(* CODESYS project Trabalho_2.project

Project tree, tasks and I/O mapping:
  Device : CODESYS Control Win V3, 3S - Smart Software Solutions GmbH, order no. 305021, version 3.5.11.30
    application Application
      libraries: Standard, * (System)
      task MainTask (cyclic, interval t#20ms, priority 1) calls PLC_PRG
      program PLC_PRG [LD]
      Symbols
*)

// Device/Application/PLC_PRG
PROGRAM PLC_PRG
VAR
	M0_1: BOOL;
	M0_0: BOOL;
	M0_2: BOOL;
	OCIOSO: BOOL;
	B_ON: BOOL;
	T01: BOOL;
	ET02: BOOL;
	A: BOOL;
	B: BOOL;
	T02: BOOL;
	ET03: BOOL;
	T03: BOOL;
	ET04: BOOL;
	T04: BOOL;
	ET05: BOOL;
	C: BOOL;
	Cont_Blocos: CTU;
	Zera_Cont: BOOL;
	Timer_Roletada: TON;
	TR: TIME;
	VOID: BOOL;
	T05: BOOL;
	T06: BOOL;
	ET06: BOOL;
	E01: BOOL;
	E02: BOOL;
	E03: BOOL;
	EB: BOOL;
	Pist_Retraido: BOOL;
	Presenca_Balanca: BOOL;
	ET07: BOOL;
	PESO: REAL;
	AUXILIAR: BOOL;
	T07: BOOL;
	TIMER_VOID: BOOL;
	T08: BOOL;
	ET08: BOOL;
	TON_0: TON;
	TIMER_TO_SEPARATION: TIME;
	EP: BOOL;
	ET09: BOOL;
	ET10: BOOL;
	ET11: BOOL;
	EM: BOOL;
	PISTAO: BOOL;
	SENSOR_PLASTICO: BOOL;
	T09: BOOL;
	TON_1: TON;
	RESET_PLASTICO: TIME;
	EP_OFF: BOOL;
	T10: BOOL;
	T11: BOOL;
	TON_2: TON;
	RESET_METAL: TIME;
	EM_OFF: BOOL;
	SENSOR_METAL: BOOL;
	VALOR: INT;
	_PESP: REAL;
	TEMPO_09: TON;
	TEMP1: TIME;
	TEMPO_11: TON;
	TEMP2: TIME;
	TIMER_BALANCA: TOF;
	TB: TIME;
	SALARIBA: BOOL;
	TIMER_BALANCA_OFF: TON;
	TIMER_BALAN: TON;
	A_OFF: TON;
	TOF_0: TOF;
	LIGADO: BOOL;
	OFF: BOOL;
	B_OFF: BOOL;
	LED_BOTAO: BOOL;
	TG: BOOL;
	BOTAO_RED: BOOL;
	TORRE_RED: BOOL;
	BOTAO_YELLOW: BOOL;
	TORRE_YELLOW: BOOL;
	EMERGENCIA: BOOL;
	CTU_0: CTU;
	SAIDA_PLASTICO: WORD;
	CTU_1: CTU;
	SAIDA_METAL: WORD;
	TOF_1: TOF;
	ABC: TIME;
	TOF_2: TOF;
	DEF: TIME;
	DESLIGA_ESTEIRAS: BOOL;
END_VAR
VAR // added by the converter: edge detectors and wires of the graphical bodies
    _w1, _w2, _w3 : BOOL;
END_VAR

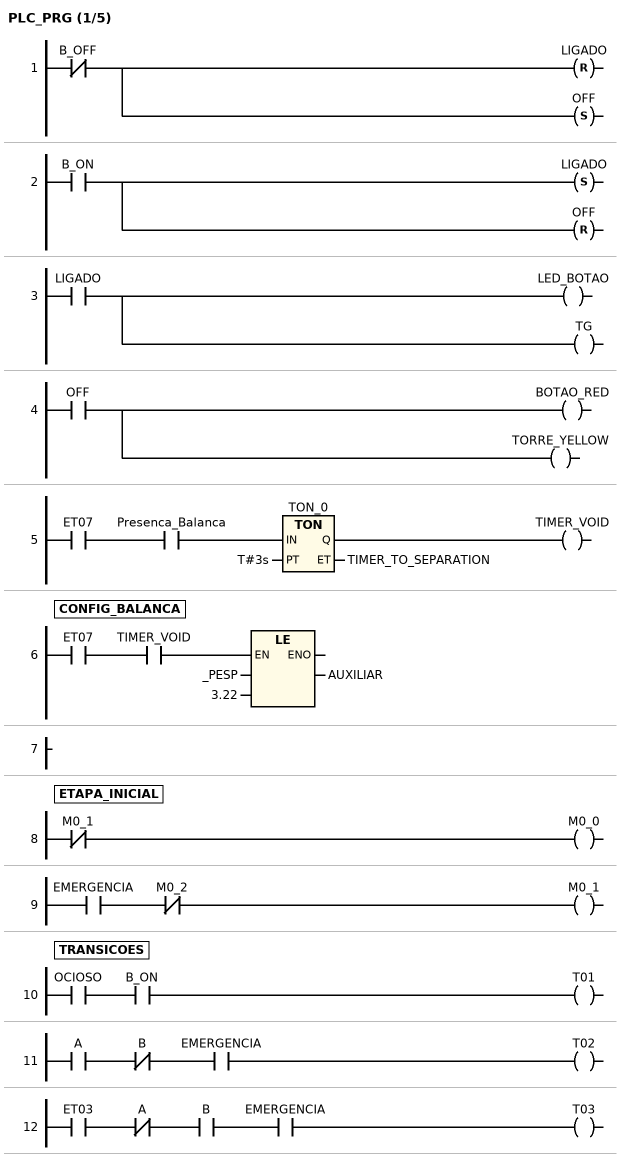
// NETWORK 1
_w1 := NOT B_OFF;
LIGADO R= _w1;
OFF S= _w1;

// NETWORK 2
LIGADO S= B_ON;
OFF R= B_ON;

// NETWORK 3
LED_BOTAO := LIGADO;
TG := LIGADO;

// NETWORK 4
BOTAO_RED := OFF;
TORRE_YELLOW := OFF;

// NETWORK 5
TON_0(IN := ET07 AND Presenca_Balanca, PT := T#3s, ET => TIMER_TO_SEPARATION); // TON
TIMER_VOID := TON_0.Q;

// NETWORK 6
CONFIG_BALANCA:
IF ET07 AND TIMER_VOID THEN AUXILIAR := _PESP <= 3.22; END_IF

// NETWORK 7

// NETWORK 8
ETAPA_INICIAL:
M0_0 := NOT M0_1;

// NETWORK 9
M0_1 := EMERGENCIA AND NOT M0_2;

// NETWORK 10
TRANSICOES:
T01 := OCIOSO AND B_ON;

// NETWORK 11
T02 := A AND NOT B AND EMERGENCIA;

// NETWORK 12
T03 := ET03 AND NOT A AND B AND EMERGENCIA;

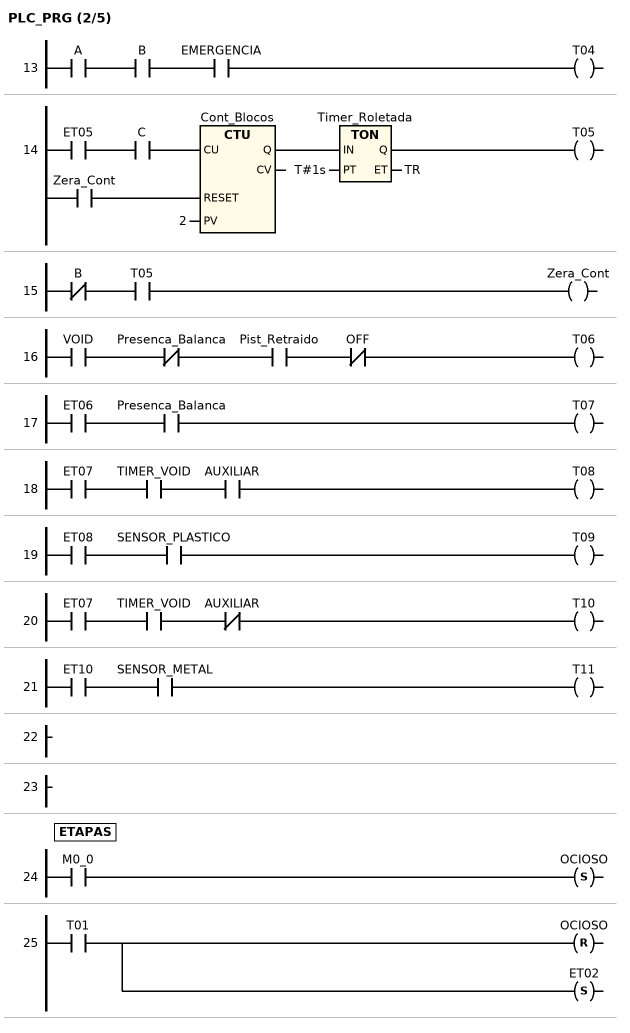
// NETWORK 13
T04 := A AND B AND EMERGENCIA;

// NETWORK 14
Cont_Blocos(CU := ET05 AND C, RESET := Zera_Cont, PV := 2); // CTU
Timer_Roletada(IN := Cont_Blocos.Q, PT := T#1s, ET => TR); // TON
T05 := Timer_Roletada.Q;

// NETWORK 15
Zera_Cont := NOT B AND T05;

// NETWORK 16
T06 := VOID AND NOT Presenca_Balanca AND Pist_Retraido AND NOT OFF;

// NETWORK 17
T07 := ET06 AND Presenca_Balanca;

// NETWORK 18
T08 := ET07 AND TIMER_VOID AND AUXILIAR;

// NETWORK 19
T09 := ET08 AND SENSOR_PLASTICO;

// NETWORK 20
T10 := ET07 AND TIMER_VOID AND NOT AUXILIAR;

// NETWORK 21
T11 := ET10 AND SENSOR_METAL;

// NETWORK 22

// NETWORK 23

// NETWORK 24
ETAPAS:
OCIOSO S= M0_0;

// NETWORK 25
OCIOSO R= T01;
ET02 S= T01;

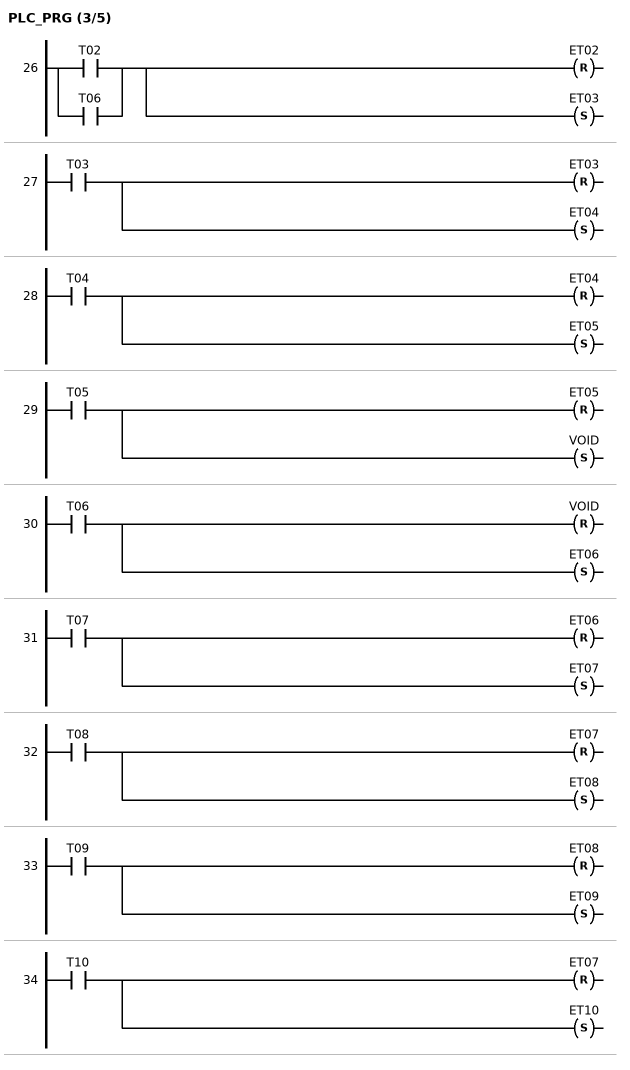
// NETWORK 26
_w2 := T02 OR T06;
ET02 R= _w2;
ET03 S= _w2;

// NETWORK 27
ET03 R= T03;
ET04 S= T03;

// NETWORK 28
ET04 R= T04;
ET05 S= T04;

// NETWORK 29
ET05 R= T05;
VOID S= T05;

// NETWORK 30
VOID R= T06;
ET06 S= T06;

// NETWORK 31
ET06 R= T07;
ET07 S= T07;

// NETWORK 32
ET07 R= T08;
ET08 S= T08;

// NETWORK 33
ET08 R= T09;
ET09 S= T09;

// NETWORK 34
ET07 R= T10;
ET10 S= T10;

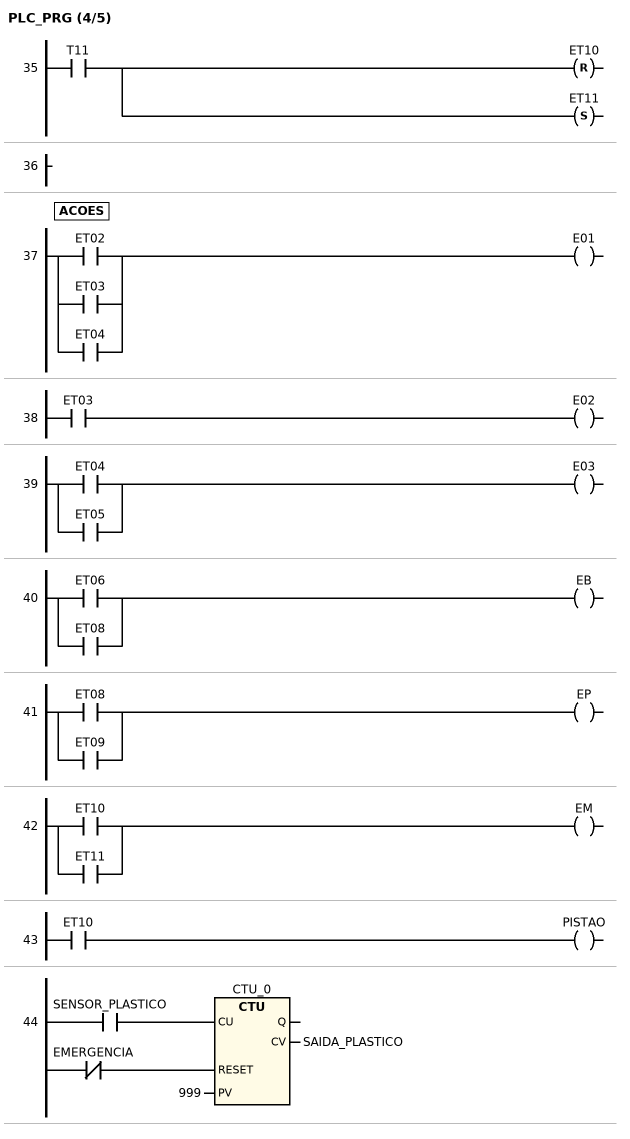
// NETWORK 35
ET10 R= T11;
ET11 S= T11;

// NETWORK 36

// NETWORK 37
ACOES:
E01 := ET02 OR ET03 OR ET04;

// NETWORK 38
E02 := ET03;

// NETWORK 39
E03 := ET04 OR ET05;

// NETWORK 40
EB := ET06 OR ET08;

// NETWORK 41
EP := ET08 OR ET09;

// NETWORK 42
EM := ET10 OR ET11;

// NETWORK 43
PISTAO := ET10;

// NETWORK 44
CTU_0(CU := SENSOR_PLASTICO, RESET := NOT EMERGENCIA, PV := 999, CV => SAIDA_PLASTICO); // CTU

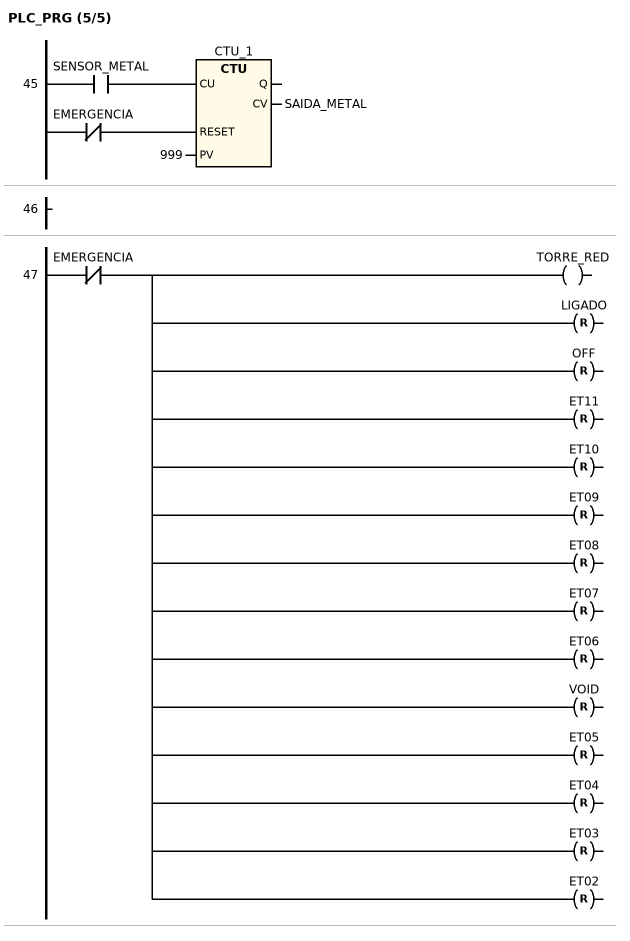
// NETWORK 45
CTU_1(CU := SENSOR_METAL, RESET := NOT EMERGENCIA, PV := 999, CV => SAIDA_METAL); // CTU

// NETWORK 46

// NETWORK 47
_w3 := NOT EMERGENCIA;
TORRE_RED := _w3;
LIGADO R= _w3;
OFF R= _w3;
ET11 R= _w3;
ET10 R= _w3;
ET09 R= _w3;
ET08 R= _w3;
ET07 R= _w3;
ET06 R= _w3;
VOID R= _w3;
ET05 R= _w3;
ET04 R= _w3;
ET03 R= _w3;
ET02 R= _w3;

END_PROGRAM
